(*
SPDX-FileCopyrightText: © 2026 Oleksandr Tiutyk <trofimich@gmail.com>
SPDX-License-Identifier: MIT
License: https://opensource.org/license/mit
*)

(*!
<summary>Writes diagnostics through TwinCAT EventLogger and expands aggregate exceptions into entries.</summary>
<description>
Provide one live event definition per category with a message placeholder {0}; the native event definition
determines event identity and severity. Constructor arguments are copied, not borrowed. No later
configuration API or native online-change handoff is provided. Keep initialization/destruction separate
from application calls; derived implementations must preserve these lifetime and no-throw guarantees.
Use this backend for TwinCAT EventLogger events with structured source information when logging errors and
exceptions directly. Use one task for direct calls on each instance without same-instance reentry; concurrent use of its internal
FB_TcEventLogger has no established guarantee here. For callers in multiple tasks, use QueuedLogger and let
only its owner task access this backend; do not bypass the wrapper with concurrent direct calls. QueuedLogger
forwards text records, so exception source is included in text rather than the structured source field, and
backend-specific aggregate formatting is not preserved. Execute performs no cyclic work. Exception logging
accepts IReadOnlyException and reads borrowed diagnostics without transferring ownership. Implementations must
not retain exception references beyond their task cleanup. Numbered messages preserve the number and truncate
oversized text to ERROR_MESSAGE capacity with a final ellipsis. TryLog methods must satisfy the no-throw
contract even when called directly, without LogManager. Does not propagate exceptions, including failures
while reading or formatting diagnostics and calling the backend; returns FALSE instead. Already emitted
entries are not rolled back, so FALSE may follow partial output. Caught exceptions are not logged again. The
fatal allocation latch is preserved for RaiseIfAllocationFailed at the task boundary outside recoverable
handlers.
</description>
*)

{attribute 'no_explicit_call' := 'do not call this function block directly'}
FUNCTION_BLOCK EventLogger EXTENDS TOF_Core.Object IMPLEMENTS TOF_Core.ILogger
VAR_STAT
	//! <summary>Static type metadata shared by instances without reading mutable instance state.</summary>
	{attribute 'hide'} 
	_ClassName : STRING := __POUNAME();
END_VAR
VAR
	
	_EventLogger : Tc3_EventLogger.FB_TcEventLogger;
	
	_DebugEventType : Global.TcEventEntry;
	_InformationEventType : Global.TcEventEntry;
	_WarningEventType : Global.TcEventEntry;
	_ErrorEventType : Global.TcEventEntry;
	_CriticalErrorEventType : Global.TcEventEntry;	
END_VAR

(*!
<summary>Provides the concrete logger type name.</summary>
<description>
Returns borrowed read-only initialized static storage. Reading has no side effects or exceptions.
Do not modify the referenced metadata; initialized storage is available before base initialization.
</description>
*)
{attribute 'monitoring' := 'call'}
PROPERTY ClassName : REFERENCE TO STRING
GET
ClassName REF= _ClassName;
END_GET
END_PROPERTY

(*!
<summary>Completes without work because this logger has no cyclic processing.</summary>
<description>Does not raise exceptions.</description>
*)
METHOD Execute
// EventLogger has no cyclic work
END_METHOD

(*!
<summary>FB_Init is always available implicitly and it is used primarily for initialization.</summary>
<description>
The return value is not evaluated. Assigns and retains event definitions for each severity category.
</description>
<param name="debugEventType">Event entry used for DEBUG category.</param>
<param name="informationEventType">Event entry used for INFORMATION category.</param>
<param name="warningEventType">Event entry used for WARNING category.</param>
<param name="errorEventType">Event entry used for ERROR category.</param>
<param name="criticalErrorEventType">Event entry used for CRITICAL_ERROR category.</param>
*)
METHOD FB_Init: BOOL
VAR_INPUT
	bInitRetains : BOOL; // TRUE: the retain variables are initialized (reset warm / reset cold)
	bInCopyCode : BOOL;  // TRUE: the instance will be copied to the copy code afterward (online change)
	debugEventType : Global.TcEventEntry;
	informationEventType : Global.TcEventEntry;
	warningEventType : Global.TcEventEntry;
	errorEventType : Global.TcEventEntry;
	criticalErrorEventType : Global.TcEventEntry;
END_VAR
_DebugEventType := debugEventType;	
_InformationEventType := informationEventType;
_WarningEventType := warningEventType;
_ErrorEventType := errorEventType;
_CriticalErrorEventType := criticalErrorEventType;
END_METHOD

(*!
<summary>Sends a diagnostic with its source and optional message number.</summary>
<description>
When a number is supplied, preserves the number prefix and as much message text as fits ERROR_MESSAGE.
Truncated text ends with U+2026. Formatting uses local storage and does not raise a size-overflow exception.
Returns FALSE for an unsupported category or failed send.
Contains formatting and native exceptions in this frame so local native FB instances exit normally.
Returns FALSE when fatal allocation state is observed before work or after nested calls. The latch remains
set for the caller's task boundary; already accepted or emitted records are not rolled back.
</description>
*)
METHOD PROTECTED InternalTryLogMessage : BOOL
VAR_INPUT
	category : TOF_Core.LOG_CATEGORY;	
END_VAR
VAR_IN_OUT CONSTANT
	message : TOF_Core.ERROR_MESSAGE;
END_VAR
VAR_INPUT
	source : Tc2_System.T_MaxString;
	messageNumber : REFERENCE TO ULINT := 0;
END_VAR
VAR	
	sourceInfo : Tc3_EventLogger.FB_TcSourceInfo;
	arguments : Tc3_EventLogger.FB_TcArguments;
	messageWithNumber : TOF_Core.ERROR_MESSAGE;
	methodResult : HRESULT;
END_VAR
__TRY

	IF TOF_Core.DynamicMemoryManager.HasAllocationFailed THEN
		RETURN;
	END_IF

	sourceInfo.sName := source;

	IF __ISVALIDREF(messageNumber) THEN
		messageWithNumber := TOF_Core.WideStrings.Concat255(
			TO_WSTRING(TOF_Core.Exceptions.MESSAGE_NUMBER_PREFIX),
			TO_WSTRING(messageNumber),
			TO_WSTRING(TOF_Core.Exceptions.MESSAGE_NUMBER_SUFFIX)
		);
		TOF_Core.WideStrings.AppendFit(targetString := messageWithNumber, sourceString := message);
		arguments.AddWString(value := messageWithNumber);
	ELSE
		arguments.AddWString(value := message);
	END_IF

	IF TOF_Core.DynamicMemoryManager.HasAllocationFailed THEN
		RETURN;
	END_IF

	CASE category OF
		TOF_Core.LOG_CATEGORY.DEBUG:
			methodResult := _EventLogger.SendMessageEx(
				stEventEntry := _DebugEventType,
				ipSourceInfo := sourceInfo,
				nTimeStamp := 0,
				ipArguments := arguments
			);

		TOF_Core.LOG_CATEGORY.INFORMATION:
			methodResult := _EventLogger.SendMessageEx(
				stEventEntry := _InformationEventType,
				ipSourceInfo := sourceInfo,
				nTimeStamp := 0,
				ipArguments := arguments
			);

		TOF_Core.LOG_CATEGORY.WARNING:
			methodResult := _EventLogger.SendMessageEx(
				stEventEntry := _WarningEventType,
				ipSourceInfo := sourceInfo,
				nTimeStamp := 0,
				ipArguments := arguments
			);

		TOF_Core.LOG_CATEGORY.ERROR:
			methodResult := _EventLogger.SendMessageEx(
				stEventEntry := _ErrorEventType,
				ipSourceInfo := sourceInfo,
				nTimeStamp := 0,
				ipArguments := arguments
			);

		TOF_Core.LOG_CATEGORY.CRITICAL_ERROR:
			methodResult := _EventLogger.SendMessageEx(
				stEventEntry := _CriticalErrorEventType,
				ipSourceInfo := sourceInfo,
				nTimeStamp := 0,
				ipArguments := arguments
			);

		ELSE
			Tc2_System.ADSLOGSTR(
				msgCtrlMask := Tc2_System.Global_Variables.ADSLOG_MSGTYPE_ERROR OR Tc2_System.Global_Variables.ADSLOG_MSGTYPE_LOG,
				msgFmtStr := Tc2_Standard.CONCAT(STR1 := 'Unsupported log category ', STR2 := TO_STRING(category)),
				strArg := ''
			);

			RETURN;
	END_CASE

	IF TOF_Core.DynamicMemoryManager.HasAllocationFailed THEN
		RETURN;
	END_IF

	IF Tc3_Module.FAILED(hr := methodResult) THEN
		Tc2_System.ADSLOGSTR(
			msgCtrlMask := Tc2_System.Global_Variables.ADSLOG_MSGTYPE_ERROR OR Tc2_System.Global_Variables.ADSLOG_MSGTYPE_LOG,
			msgFmtStr := Tc2_Standard.CONCAT(
				STR1 := 'FB_TcMessage creation failed with HRESULT = ',
				STR2 := TO_STRING(methodResult)
			),
			strArg := ''
		);

		RETURN;
	END_IF

	InternalTryLogMessage := TRUE;

	IF TOF_Core.DynamicMemoryManager.HasAllocationFailed THEN
		InternalTryLogMessage := FALSE;
	END_IF

__CATCH
	// Contain failure before local native argument/source objects leave this frame.
	InternalTryLogMessage := FALSE;
__ENDTRY
END_METHOD

(*!
<summary>Borrows the library namespace.</summary>
<description>
Read-only compiler-initialized storage; do not modify the referenced text.
</description>
*)
{attribute 'monitoring' := 'call'}
PROPERTY NamespaceName : REFERENCE TO STRING
GET
NamespaceName REF= CurrentNamespace.Name;
END_GET
END_PROPERTY

(*!
<summary>Reports the size of this concrete event logger instance.</summary>
<description>
The result includes embedded native state but excludes allocations owned internally by native services.
</description>
*)
{attribute 'monitoring' := 'call'}
PROPERTY SelfSize : ULINT
GET
SelfSize := XSIZEOF(THIS^);
END_GET
END_PROPERTY

(*!
<summary>Attempts to log a borrowed error without propagating exceptions.</summary>
<description>
Borrows inputs only for the call. TRUE reports backend acceptance, not guaranteed durable storage. Does not
propagate exceptions, including failures while reading or formatting diagnostics and calling the backend;
returns FALSE instead. Already emitted entries are not rolled back, so FALSE may follow partial output. Caught
exceptions are not logged again. The fatal allocation latch is preserved for RaiseIfAllocationFailed at the
task boundary outside recoverable handlers.
Returns FALSE when fatal allocation state is observed before work or after nested calls. The latch remains
set for the caller's task boundary; already accepted or emitted records are not rolled back.
</description>
*)
METHOD TryLogError : BOOL
VAR_INPUT
	error : REFERENCE TO TOF_Core.ERROR;
	messageNumber : REFERENCE TO ULINT := 0;
END_VAR
VAR
	message : TOF_Core.ERROR_MESSAGE;
END_VAR
__TRY

	IF TOF_Core.DynamicMemoryManager.HasAllocationFailed THEN
		RETURN;
	END_IF

	IF NOT __ISVALIDREF(error) THEN
		RETURN;
	END_IF

	message := error.ToString(
		sourceDisplayMode := TOF_Core.ERROR_SOURCE_DISPLAY_MODE.HIDDEN,
		timestampDisplayMode := TOF_Core.TIMESTAMP_DISPLAY_MODE.HIDDEN
	);

	IF TOF_Core.DynamicMemoryManager.HasAllocationFailed THEN
		RETURN;
	END_IF

	TryLogError := InternalTryLogMessage(
		category := SEL(
			error.Severity = TOF_Core.ERROR_SEVERITY.CRITICAL,
			TOF_Core.LOG_CATEGORY.ERROR,
			TOF_Core.LOG_CATEGORY.CRITICAL_ERROR
		),
		message := message,
		source := error.GetSource(appendRootSource := TRUE),
		messageNumber := messageNumber
	);

	IF TOF_Core.DynamicMemoryManager.HasAllocationFailed THEN
		TryLogError := FALSE;
	END_IF

__CATCH
	TryLogError := FALSE;
__ENDTRY
END_METHOD

(*!
<summary>Attempts to log diagnostic information from a read-only exception view.</summary>
<description>
Borrows the exception for the call without clearing it or taking ownership. The exception and its inner causes
must remain live and form an acyclic graph while their diagnostics are read. Nonempty aggregates produce
separate entries in stored order, sharing the optional request number. Nonfatal FALSE does not suppress later
entries; a thrown diagnostic failure or observed terminal allocation state stops further processing. Logging does not extend their lifetime. Does not propagate
exceptions, including failures while reading or formatting diagnostics and calling the backend; returns FALSE
instead. Already emitted entries are not rolled back, so FALSE may follow partial output. Caught exceptions
are not logged again. The fatal allocation latch is preserved for RaiseIfAllocationFailed at the task boundary
outside recoverable handlers.
Returns FALSE when fatal allocation state is observed before work or after nested calls. The latch remains
set for the caller's task boundary; already accepted or emitted records are not rolled back.
</description>
<param name="exception">Exception view to read; null is ignored.</param>
<param name="severity">Severity used to select the log category.</param>
*)
METHOD TryLogException : BOOL
VAR_INPUT
	exception : TOF_Core.IReadOnlyException;
	severity : TOF_Core.ERROR_SEVERITY;
	messageNumber : REFERENCE TO ULINT := 0;
END_VAR
VAR
	message : TOF_Core.ERROR_MESSAGE;
	aggregateException : TOF_Core.IAggregateException;
	innerExceptionCount : UINT;
	i : DINT;
END_VAR
__TRY

	IF TOF_Core.DynamicMemoryManager.HasAllocationFailed THEN
		RETURN;
	END_IF

	IF exception = 0 THEN
		RETURN;
	END_IF

	IF __QUERYINTERFACE(exception, aggregateException) THEN
		innerExceptionCount := aggregateException.InnerExceptionCount;
	END_IF

	IF TOF_Core.DynamicMemoryManager.HasAllocationFailed THEN
		RETURN;
	END_IF

	IF innerExceptionCount = 0 THEN
		message := exception.GetMessage(showSource := FALSE, timestampDisplayMode := TOF_Core.TIMESTAMP_DISPLAY_MODE.LOCAL);

		IF TOF_Core.DynamicMemoryManager.HasAllocationFailed THEN
			RETURN;
		END_IF

		TryLogException := InternalTryLogMessage(
			category := SEL(severity = TOF_Core.ERROR_SEVERITY.CRITICAL, TOF_Core.LOG_CATEGORY.ERROR, TOF_Core.LOG_CATEGORY.CRITICAL_ERROR),
			message := message,
			source := exception.GetSourceDescription(),
			messageNumber := messageNumber
		);
	ELSE
		TryLogException := TRUE;

		FOR i := 0 TO TO_DINT(innerExceptionCount) - 1 DO

			IF TOF_Core.DynamicMemoryManager.HasAllocationFailed THEN
				TryLogException := FALSE;
				RETURN;
			END_IF

			TryLogException := TryLogException AND THIS^.TryLogException(
				exception := aggregateException.GetInnerException(index := i),
				severity := severity,
				messageNumber := messageNumber
			);

			IF TOF_Core.DynamicMemoryManager.HasAllocationFailed THEN
				TryLogException := FALSE;
				RETURN;
			END_IF

		END_FOR

	END_IF

	IF TOF_Core.DynamicMemoryManager.HasAllocationFailed THEN
		TryLogException := FALSE;
	END_IF

__CATCH
	TryLogException := FALSE;
__ENDTRY
END_METHOD

(*!
<summary>Attempts to log borrowed message text without propagating exceptions.</summary>
<description>
Borrows inputs only for the call. TRUE reports backend acceptance, not guaranteed durable storage. Does not
propagate exceptions, including failures while reading or formatting diagnostics and calling the backend;
returns FALSE instead. Already emitted entries are not rolled back, so FALSE may follow partial output. Caught
exceptions are not logged again. The fatal allocation latch is preserved for RaiseIfAllocationFailed at the
task boundary outside recoverable handlers.
Returns FALSE when fatal allocation state is observed before work or after nested calls. The latch remains
set for the caller's task boundary; already accepted or emitted records are not rolled back.
</description>
*)
METHOD TryLogMessage : BOOL
VAR_INPUT
	category : TOF_Core.LOG_CATEGORY;	
END_VAR
VAR_IN_OUT CONSTANT
	message : TOF_Core.ERROR_MESSAGE;
END_VAR
VAR_INPUT
	messageNumber : REFERENCE TO ULINT := 0;
END_VAR
__TRY

	IF TOF_Core.DynamicMemoryManager.HasAllocationFailed THEN
		RETURN;
	END_IF

	TryLogMessage := InternalTryLogMessage(category := category, message := message, source := '', messageNumber := messageNumber);

	IF TOF_Core.DynamicMemoryManager.HasAllocationFailed THEN
		TryLogMessage := FALSE;
	END_IF

__CATCH
	TryLogMessage := FALSE;
__ENDTRY
END_METHOD

END_FUNCTION_BLOCK

(* stored: Version 1.1.0.1
   POU EventLogger: Id {54f03143-ac47-4e1f-bf2d-cc4de4cc1513}, SpecialFunc None
   Folder Internal members: Id {eb43b981-fe0c-4384-9a7e-ded8f887a71f}
   Property ClassName: Id {8606f867-ab71-4ff0-b44a-b045271484a0}
   Get Get: Id {3237a013-9364-426b-a2dd-3913256764ad}
   Method Execute: Id {45bb9e14-c21d-4ace-9cc8-e5705603b0cc}
   Method FB_Init: Id {e52cf092-8b74-4e13-811f-db521a4e102c}
   Method InternalTryLogMessage: Id {b17f1f74-b328-47c1-a9cb-5cbdf2cd529f}
   Property NamespaceName: Id {75388737-b788-4a16-a31f-a3885f5f2749}
   Get Get: Id {751a8249-a618-42a3-8fb5-6e37489fe438}
   Property SelfSize: Id {98e9eadc-01ba-46bc-90cb-368644546c24}
   Get Get: Id {606ae824-c393-4762-992a-f3ef439dd9fb}
   Method TryLogError: Id {4a210b47-12f5-416e-800c-6b940764fae5}
   Method TryLogException: Id {1990277d-d5d3-4267-af7a-8be26122cbfe}
   Method TryLogMessage: Id {68073492-716c-4ee9-a006-f48bbbfa1f4f} *)
